// TIA Portal V17 program export: 1 tag tables, 0 data types, 0 data blocks, 9 code blocks (in call order from the OBs), 0 instance data blocks

VAR_GLOBAL   // PLC tag table "Default tag table"
END_VAR

ORGANIZATION_BLOCK "Main"   // OB1, LAD, ProgramCycle
TITLE = "Main Program Sweep (Cycle)"
{ S7_Optimized_Access := 'TRUE' }
VERSION : 0.1
// stored: AutoNumber true, IsIECCheckEnabled false, SetENOAutomatically false
   VAR_INPUT
      Initial_Call : Bool;   // Initial call of this OB
      Remanence : Bool;   // =True, if remanent data are available
   END_VAR
   VAR_TEMP
      temp_1 : Bool;
      temp_2 : Bool;
      "temp Int" : Int;
   END_VAR
   VAR_TEMP   // added for the SCL form of the ladder/FBD networks
      _w1 : Bool;
   END_VAR
BEGIN

REGION Network 1
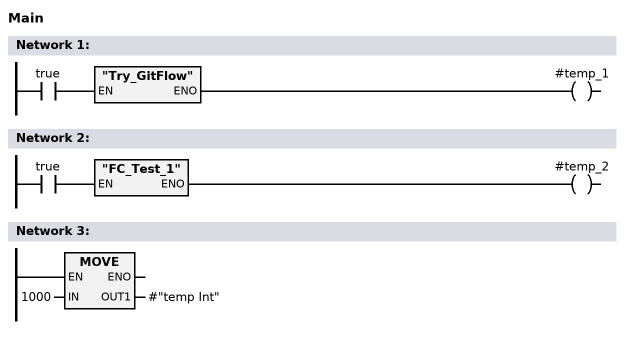
   RUNG wire#powerrail
      Contact( true )
      "Try_GitFlow"()
      Coil( #temp_1 )
   END_RUNG
   // the same network as SCL:
   "Try_GitFlow"(EN := true, ENO => #_w1);
   #temp_1 := #_w1;
END_REGION

REGION Network 2
   RUNG wire#powerrail
      Contact( true )
      "FC_Test_1"()
      Coil( #temp_2 )
   END_RUNG
   // the same network as SCL:
   "FC_Test_1"(EN := true, ENO => #_w1);
   #temp_2 := #_w1;
END_REGION

REGION Network 3
   RUNG wire#powerrail
      Move(in := 1000, out1 => #"temp Int")
   END_RUNG
   // the same network as SCL:
   #"temp Int" := 1000;
END_REGION
END_ORGANIZATION_BLOCK

FUNCTION "Try_GitFlow" : Void   // FC3, LAD
{ S7_Optimized_Access := 'TRUE' }
VERSION : 0.1
// stored: AutoNumber true, IsIECCheckEnabled false, SetENOAutomatically false, UDAEnableTagReadback false
BEGIN
END_FUNCTION

FUNCTION "FC_Test_1" : Void   // FC1, SCL
{ S7_Optimized_Access := 'TRUE' }
VERSION : 0.1
// stored: AutoNumber true, IsIECCheckEnabled false, SetENOAutomatically false, UDAEnableTagReadback false
   VAR_TEMP
      temp_1 : Bool;
      temp_2 : Bool;
      temp_git : Bool;
   END_VAR
BEGIN
   // version branch evo
   IF #temp_1 THEN
       // Statement section IF
       #temp_2 := true;
   END_IF;

   // use XML export to use ACT + created branch
END_FUNCTION

FUNCTION "FC_SubFun_1" : Void   // FC4, LAD
{ S7_Optimized_Access := 'TRUE' }
VERSION : 0.1
// stored: AutoNumber true, IsIECCheckEnabled false, SetENOAutomatically false, UDAEnableTagReadback false
BEGIN
END_FUNCTION

FUNCTION "FC_SubFun_2" : Void   // FC4, LAD
{ S7_Optimized_Access := 'TRUE' }
VERSION : 0.1
// stored: AutoNumber true, IsIECCheckEnabled false, SetENOAutomatically false, UDAEnableTagReadback false
BEGIN
END_FUNCTION

FUNCTION "FC_SubFun_A" : Void   // FC4, LAD
{ S7_Optimized_Access := 'TRUE' }
VERSION : 0.1
// stored: AutoNumber true, IsIECCheckEnabled false, SetENOAutomatically false, UDAEnableTagReadback false
BEGIN
END_FUNCTION

FUNCTION "FC_SubFun_B" : Void   // FC4, LAD
{ S7_Optimized_Access := 'TRUE' }
VERSION : 0.1
// stored: AutoNumber true, IsIECCheckEnabled false, SetENOAutomatically false, UDAEnableTagReadback false
BEGIN
END_FUNCTION

FUNCTION "FC_Test_2" : Void   // FC2, LAD
{ S7_Optimized_Access := 'TRUE' }
VERSION : 0.1
// stored: AutoNumber true, IsIECCheckEnabled false, SetENOAutomatically false, UDAEnableTagReadback false
   VAR_TEMP
      temp_1 : Bool;
   END_VAR
BEGIN

REGION Network 1
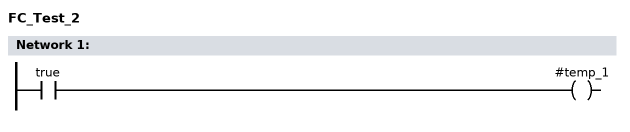
   RUNG wire#powerrail
      Contact( true )
      Coil( #temp_1 )
   END_RUNG
   // the same network as SCL:
   #temp_1 := true;
END_REGION
END_FUNCTION

FUNCTION "FC_Test_3" : Void   // FC4, LAD
{ S7_Optimized_Access := 'TRUE' }
VERSION : 0.1
// stored: AutoNumber true, IsIECCheckEnabled false, SetENOAutomatically false, UDAEnableTagReadback false
BEGIN
END_FUNCTION
